{attribute 'qualified_only'}
{attribute 'strict'}
(* Motion-generation independent jog mode.
   Mapped onto Tc2_MC2.E_JogMode / Tc3_Mc3Ptp.EJogMode by the concrete axis. *)
TYPE E_AxisJogMode : (
		Slow := 0,
		Fast := 1
	) DINT;
END_TYPE

(* stored: Version 1.1.0.1, ProductVersion 3.1.4026.20
   DUT E_AxisJogMode: Id {4b39cb50-23f6-4cce-9c25-5daecbf6b9cb} *)
